FUNCTION_BLOCK ABSTRACT FM_Maschine EXTENDS FD_Device 
VAR_INPUT
END_VAR
VAR_OUTPUT
END_VAR
VAR
	// Global child status
	bAllChildsReady 					: BOOL;
	bAllChildsHomed 					: BOOL;
	bAllChildsDone  					: BOOL;
	bAnyChildBusy   					: BOOL;
	bAnyChildError  					: BOOL;
	// Internal command state
	eLastChildCmdState 				: E_CmdState;
	
	// Hmi Variable
	stHMI 										: ST_MaschineHMI;
END_VAR


SUPER^();

mVisu();
// Update global child status every PLC cycle
mUpdateChildsState();

IF SequenceBusy THEN
    mSequence(TRUE);
END_IF

//FB_Init ist immer implizit verfügbar und wird primär für die Initialisierung verwendet.
//Der Rückgabewert wird nicht ausgewertet. Für gezielte Einflussnahme können Sie
//die Methoden explizit deklarieren und darin mit dem Standard-Initialisierungscode 
//zusätzlichen Code bereitstellen. Sie können den Rückgabewert auswerten.
METHOD FB_Init: BOOL
VAR_INPUT    
	bInitRetains					: BOOL; 					// TRUE: Die Retain-Variablen werden initialisiert (Reset warm / Reset kalt)    
	bInCopyCode						: BOOL;  					// TRUE: Die Instanz wird danach in den Kopiercode kopiert (Online-Change)
	
	I_Name                : STRING;         //  Name
	I_ID                  : UINT;           // ID
  I_itfOwner					  : ITF_Owner;      // owner 
END_VAR
END_METHOD

METHOD mAutomatic : E_CmdState
VAR_INPUT
	I_bExecute	: BOOL;
END_VAR

// Call mAutomatic in Base
SUPER^.mAutomatic(I_bExecute);

// Machine can only go AUTO if all child devices are homed
mUpdateChildsState();

IF NOT bAllChildsHomed 
	THEN
    mAutomatic := E_CmdState.NotReady;
    RETURN;
END_IF
END_METHOD

METHOD mCheckAllChildsReady : Bool
VAR_INPUT
END_VAR
END_METHOD

METHOD mHome : E_CmdState
VAR_INPUT
	I_bExecute	: BOOL;
END_VAR

mHome := SUPER^.mHome(I_bExecute);

// If generic checks failed -> exit
IF mHome <> E_CmdState.Busy THEN RETURN; END_IF

// Machine-specific preparation
mUpdateChildsState();

// verify children available before homing
IF bAnyChildError 
	THEN
    mHome := E_CmdState.Error;
    RETURN;
END_IF
END_METHOD

METHOD mReset : BOOL
VAR_INPUT
END_VAR
VAR
	L_uiIndex   : UINT;
END_VAR

// Reset own machine state from parent class
//==================================================
SUPER^.mReset();

// Reset all register child devices
//==================================================
FOR L_uiIndex := 1 TO uiChildsCount DO
	aitfChilds[L_uiIndex].mReset();
END_FOR

// Reset machine supervision flags
//==================================================
bAllChildsReady 							:= FALSE;
bAllChildsHomed 							:= FALSE;
bAllChildsDone  							:= FALSE;
                							
bAnyChildBusy   							:= FALSE;
bAnyChildError  							:= FALSE;

// Reset machine sequence
//==================================================
SequenceID 										:= C_SeqStep_Idle;
              								
bSequenceBusy 								:= FALSE;
bSequenceDone 								:= FALSE;
              								
bReady 												:= FALSE;
bHomed 												:= FALSE;

// Reset machine mode
//==================================================
Mode 													:= E_Mode.IDLE;

// Reset successful
//==================================================
mReset := TRUE;
END_METHOD

METHOD mSequence : E_CmdState
VAR_INPUT
	I_bExecute				: BOOL;
END_VAR

VAR
    eCmd 						: E_CmdState;
END_VAR

// Generic pre-check from parent
mSequence := SUPER^.mSequence(I_bExecute := I_bExecute);

IF mSequence <> E_CmdState.Busy THEN
    RETURN;
END_IF

// Update child status before sequence logic
mUpdateChildsState();

IF bAnyChildError THEN
    SequenceID := C_SeqStep_Error;
END_IF

CASE SequenceID OF
    C_SeqStep_Start:
        CASE Mode OF
        	E_Mode.Homing:
        	    eCmd 	:= mSetChildMode(E_Mode.Homing);
        	E_Mode.Auto:
        	    eCmd 	:= mSetChildMode(E_Mode.Auto);
        	E_Mode.Service:
        	    eCmd 	:= mSetChildMode(E_Mode.Service);
        END_CASE
    	SequenceID := 10;
      mSequence := E_CmdState.Busy;

    10:
        // Wait until all child devices finish their requested command
        mUpdateChildsState();

        IF bAnyChildError THEN
            SequenceID := C_SeqStep_Error;

        ELSIF NOT bAnyChildBusy THEN
            SequenceID := C_SeqStep_Done;
        END_IF
        mSequence := E_CmdState.Busy;
				
    C_SeqStep_Done:
    	bSequenceBusy := FALSE;
    	bSequenceDone := TRUE;
    	
    	IF Mode = E_Mode.Homing 
				THEN
    	    bHomed := TRUE;
    	END_IF
    	
    	bReady := TRUE;
    	SequenceID := C_SeqStep_Idle;
    	
    	mSequence := E_CmdState.Succeeded;
    	
    C_SeqStep_Error:
    	bError := TRUE;
    	bSequenceBusy := FALSE;
    	bSequenceDone := FALSE;
    	
    	mSequence := E_CmdState.Error;
    	
    ELSE
        SequenceID := C_SeqStep_Error;
        mSequence := E_CmdState.Error;

END_CASE
END_METHOD

METHOD PROTECTED mSetChildMode  : E_CmdState
VAR_INPUT
	I_eMode 		: E_Mode;
END_VAR

VAR
	uiIndex 		: UINT;
  eCmd 				: E_CmdState;
END_VAR

mSetChildMode := E_CmdState.Succeeded;

// Send requested mode command to all child devices
FOR uiIndex := 1 TO uiChildsCount DO
	CASE I_eMode OF
  	E_Mode.Homing:
  		eCmd 			    := aitfChilds[uiIndex].mHome(TRUE);
  	E_Mode.Auto:
  		eCmd 			    := aitfChilds[uiIndex].mAutomatic(TRUE);
  	E_Mode.Service:
  		eCmd 			    := aitfChilds[uiIndex].mService(TRUE);			
		E_Mode.Idle:
  		eCmd 			    := aitfChilds[uiIndex].mStop(TRUE);
  	E_Mode.Error:
  		eCmd 			    := aitfChilds[uiIndex].mAbort(TRUE);
  END_CASE

    // If one child is busy, global command is still busy
	IF eCmd = E_CmdState.Busy 
		THEN
	    mSetChildMode  := E_CmdState.Busy;
	END_IF
	 
	// If one child has error, global command is error
	IF (eCmd = E_CmdState.Error) OR (eCmd = E_CmdState.NotReady) 
  	THEN
	    mSetChildMode  := eCmd;
	    RETURN;
	END_IF
END_FOR
END_METHOD

METHOD mStop : E_CmdState
VAR_INPUT
	I_bExecute	: BOOL;
END_VAR

// Stop machine base status
SUPER^.mStop(I_bExecute);

// Stop all child devices
 //StopChilds();
END_METHOD

METHOD PROTECTED mStopChilds  : E_CmdState
VAR_INPUT
END_VAR

VAR
    uiIndex 				: UINT;
    eCmd 						: E_CmdState;
END_VAR

mStopChilds := E_CmdState.Succeeded;

// Stop all child devices
FOR uiIndex := 1 TO uiChildsCount DO
	eCmd := aitfChilds[uiIndex].mStop(TRUE);
	
	IF eCmd = E_CmdState.Busy 
		THEN
	    mStopChilds := E_CmdState.Busy;
	END_IF
	
	IF eCmd = E_CmdState.Error 
		THEN
	    mStopChilds := E_CmdState.Error;
	    RETURN;
    END_IF
END_FOR
END_METHOD

METHOD PROTECTED mUpdateChildsState  : BOOL
VAR_INPUT
END_VAR
VAR
	L_uiIndex									: UINT;
	
END_VAR

// Evaluate all registered child devices
FOR L_uiIndex := 1 TO uiChildsCount DO

    IF aitfChilds[L_uiIndex].Error THEN
        bAnyChildError := TRUE;
    END_IF

    IF aitfChilds[L_uiIndex].SequenceBusy THEN
        bAnyChildBusy := TRUE;
    END_IF

    IF NOT aitfChilds[L_uiIndex].Ready THEN
        bAllChildsReady := FALSE;
    END_IF

    IF NOT aitfChilds[L_uiIndex].Homed THEN
        bAllChildsHomed := FALSE;
    END_IF

    IF NOT aitfChilds[L_uiIndex].SequenceDone THEN
        bAllChildsDone := FALSE;
    END_IF

END_FOR

mUpdateChildsState := TRUE;
END_METHOD

METHOD mVisu : BOOL
VAR_INPUT
END_VAR

// Status to HMI
	stHMI.sName     					:= Name;
	stHMI.uiID      					:= ID;
	stHMI.bReady    					:= Ready;
	stHMI.bHomed    					:= Homed;
	stHMI.bBusy     					:= SequenceBusy;
	stHMI.bDone     					:= SequenceDone;
	stHMI.bError    					:= Error;
	stHMI.eMode     					:= Mode;
	stHMI.uiSequenceID    		:= SequenceID;
	
	// Commands from HMI
	IF stHMI.bCmdReset 
		THEN
	    mReset();
	    stHMI.bCmdReset := FALSE;
	END_IF
	
	IF stHMI.bCmdHome 
		THEN
	    stHMI.eCmdState := mHome(TRUE);
	    stHMI.bCmdHome := FALSE;
	END_IF
	
	IF stHMI.bCmdAuto 
		THEN
	    stHMI.eCmdState := mAutomatic(TRUE);
	    stHMI.bCmdAuto := FALSE;
	END_IF
	
	IF stHMI.bCmdService 
  	THEN
	    stHMI.eCmdState := mService(TRUE);
	    stHMI.bCmdService := FALSE;
	END_IF
	
	IF stHMI.bCmdStop 
		THEN
    stHMI.eCmdState := mStop(TRUE);
    stHMI.bCmdStop := FALSE;
END_IF

IF stHMI.bCmdAbort 
	THEN
    stHMI.eCmdState := mAbort(TRUE);
    stHMI.bCmdAbort := FALSE;
END_IF

mVisu := TRUE;
END_METHOD

END_FUNCTION_BLOCK

(* stored: Version 1.1.0.1, ProductVersion 3.1.4026.18
   POU FM_Maschine: Id {83e5710c-69e8-4593-a566-ae4a485f5caa}, SpecialFunc None
   Folder 01 Properties: Id {6a87ee5d-b4db-4b64-8036-f307a328febf}
   Folder 02 Methodes: Id {5561014d-7db8-4950-aa75-2604d264aa2f}
   Folder 010 _SetChild: Id {e5bea0b9-25fa-45a2-9e8c-d054885de145}
   Folder 020 OpMode: Id {85940346-4c69-4b4c-b5e9-25a708434663}
   Folder 040 Fx: Id {42cfef7c-3ff8-4651-b791-27ca4000f4e5}
   Folder 099 HMI: Id {07d2b20f-db9e-47fa-8a44-e2847c19c7af}
   Method FB_Init: Id {4d06739b-5dd6-4759-85b3-148920b74dbe}
   Method mAutomatic: Id {34b44ad0-f67d-44fe-a6ef-a7575f674d83}
   Method mCheckAllChildsReady: Id {39b8dd00-c2ac-4bef-91c5-3bcadfa4b938}
   Method mHome: Id {95927eb3-0055-4f5c-b3ae-60a81380b498}
   Method mReset: Id {5ff340bf-d875-48ce-8ee0-ba78a52617fe}
   Method mSequence: Id {d50b92a4-7563-419d-8a14-262b8f70b0f9}
   Method mSetChildMode: Id {b359a2b7-9f9a-4774-a7bb-b44d823f4f2a}
   Method mStop: Id {7eecaabd-8804-4508-8714-47321ca48c04}
   Method mStopChilds: Id {d8d10ce1-d462-401a-b1f9-a70c4c67ef67}
   Method mUpdateChildsState: Id {54b84bff-c321-4ea9-8af5-5f96b3fa3112}
   Method mVisu: Id {755d8c18-c470-42a3-9fc7-897d4f23f899} *)
